	                // Check sequence number. If it is equal or greater than 30000 reset it to 1.
	                IF #iqdi_MessageSequenceNumber < 30000
	                THEN
	                    #iqdi_MessageSequenceNumber += 1;
	                ELSE
	                    #iqdi_MessageSequenceNumber := 1;
	                END_IF;

	                #ss_NewStatusMessage[#ti_Loop_ItemStatus_FiFo].Size := #ss_NewStatusMessage[#ti_Loop_ItemStatus_FiFo].Size * #ci_ItemStatus_BodyLenght;

	                // Write parts of the header into structure.
	                #s_UDT_MessageHeader.BodyLength := #ss_NewStatusMessage[#ti_Loop_ItemStatus_FiFo].Size;
	                #s_UDT_MessageHeader.FlagRetry.%X0 := FALSE;
	                #s_UDT_MessageHeader.Group := 1;
	                #s_UDT_MessageHeader.MessageID := #ci_ItemStatus_MessageID;
	                #s_UDT_MessageHeader.SequenceNumber := #iqdi_MessageSequenceNumber;
	                #s_UDT_MessageHeader.TimeSpan := 0;

	                // Calculate the header checksum.
	                "FC_Checksum"(i_UDT_MessageHeader := #s_UDT_MessageHeader,
	                              qb_Checksum => #s_UDT_MessageHeader.Checksum);

	                // Initialize the header serialize position and convert header structure into array of bytes.
	                #sdi_SerializePosition := 0;
	                #si_HeaderSerializeStatus := Serialize(SRC_VARIABLE := #s_UDT_MessageHeader,
	                                                       DEST_ARRAY => #s_UDT_MessageArray.Bytes,
	                                                       POS := #sdi_SerializePosition);

	                FOR #ti_Loop_ItemStatus_FiFo_1 := 1 TO #ss_NewStatusMessage[#ti_Loop_ItemStatus_FiFo].Size / #ci_ItemStatus_BodyLenght DO

	                    #s_UDT_ItemStatusBody := #ss_NewStatusMessage[#ti_Loop_ItemStatus_FiFo].Body[#ti_Loop_ItemStatus_FiFo_1];

	                    // Convert message body structure into array of bytes.
	                    #si_BodySerializeStatus := Serialize(SRC_VARIABLE := #s_UDT_ItemStatusBody,
	                                                         DEST_ARRAY => #s_UDT_MessageArray.Bytes,
	                                                         POS := #sdi_SerializePosition);
	                END_FOR;

	                // Mode 'W' - Write FIFO record.
	                "FC_Fifo"(ic_Mode := 'W',
	                          qUDT_Status => #ss_Status.FIFOItemStatusStatus,
	                          qx_Error => #ss_Status.FIFOError,
	                          qx_Warning => #ss_Status.FIFOWarning,
	                          iqv_Data := #s_UDT_MessageArray,
	                          iqUDT_FifoHeader := #iq_UDT_FifoReceiveHeader_Out,
	                          iqv_DataBuffer := #iqs_FifoReceiveData_Out);
	            END_FOR;

	            #si_Counter_ItemStatus := 0;

	        END_IF;

	    END_REGION

	    REGION 3.3 Other types of messages

	        IF #si_Counter_InvalidMessageID > 0 THEN

	            FOR #ti_Loop_InvalidMessageID := 1 TO #si_Counter_InvalidMessageID DO

	                // Mode 'W' - Write FIFO record.
	                "FC_Fifo"(ic_Mode := 'W',
	                          qUDT_Status => #ss_Status.FIFOInvalidMessageIDStatus,
	                          qx_Error => #ss_Status.FIFOError,
	                          qx_Warning => #ss_Status.FIFOWarning,
	                          iqv_Data := #sa_Data_InvalidMessageID[#ti_Loop_InvalidMessageID],
	                          iqUDT_FifoHeader := #iq_UDT_FifoReceiveHeader_Out,
	                          iqv_DataBuffer := #iqs_FifoReceiveData_Out);

	            END_FOR;

	            #si_Counter_InvalidMessageID := 0;

	        END_IF;

	    END_REGION

	END_REGION



END_FUNCTION_BLOCK

